TYPE Status_MV :
(
		Normalbetrieb,
		PumpDown,
		AbtauenOben,
		AbtauenUnten
);
END_TYPE

(* stored: Version 1.1.0.1, ProductVersion 3.1.4018.5
   DUT Status_MV: Id {dfd13b30-6fe1-4769-8b5d-0022cc9cf87c} *)
